// TIA Portal project "KWT_80413" (V14)

(* hardware
DEVICE "S7-1200-Station_1"  S7-1200 Station
   slot 0: "Baugruppenträger_0"  S7-1200 Rack  Rack  V1.0
   slot 1: "PLC_1"  CPU 1212C AC/DC/Rly  6ES7 212-1BE40-0XB0  V4.2
   slot 2: "AQ 2x14BIT_1"  SM 1232 AQ2  6ES7 232-4HB32-0XB0  V2.0
   slot 3: "DI 16x24VDC_1"  6ES7 221-1BH32-0XB0  V2.0
DEVICE "HMI_1"  KTP1200 Basic PN
   slot 0: "KTP1200 Basic PN"  KTP1200 Basic PN  6AV2 123-2MB03-0AX0  14.0.1.0
   slot 1: "HMI_RT_1"  KTP1200 Basic PN  6AV2 123-2MB03-0AX0  14.0.1.0
   slot 5: "HMI_1.IE_CP_1"  PROFINET Interface  14.0.1.0
      slot 1: "PROFINET Schnittstelle_1"  PROFINET Interface
         slot 1: "Port_1"  Port
*)

// ===== PLC "PLC_1"  CPU 1212C AC/DC/Rly =====

VAR_GLOBAL   // PLC tag table "Standard-Variablentabelle"
   "System_Byte" AT %MB1 : Byte;
   "FirstScan" AT %M1.0 : Bool;
   "DiagStatusUpdate" AT %M1.1 : Bool;
   "AlwaysTRUE" AT %M1.2 : Bool;
   "AlwaysFALSE" AT %M1.3 : Bool;
   "Clock_Byte" AT %MB0 : Byte;
   "Clock_10Hz" AT %M0.0 : Bool;
   "Clock_5Hz" AT %M0.1 : Bool;
   "Clock_2.5Hz" AT %M0.2 : Bool;
   "Clock_2Hz" AT %M0.3 : Bool;
   "Clock_1.25Hz" AT %M0.4 : Bool;
   "Clock_1Hz" AT %M0.5 : Bool;
   "Clock_0.625Hz" AT %M0.6 : Bool;
   "Clock_0.5Hz" AT %M0.7 : Bool;
   "Pumpe 1" AT %Q0.0 : Bool;   // Pumpe 1, -102K1, -36K6, Werkskreislauf
   "Pumpe 2" AT %Q0.1 : Bool;   // Pumpe 2, -102K2, -38K6, Werkskreislauf
   "Pumpe 3" AT %Q0.2 : Bool;   // Pumpe 3, -102K3, -41K6, Kühlturmkreislauf
   "Pumpe 4" AT %Q0.3 : Bool;   // Pumpe 4, -102K4, -43K6, Kühlturmkreislauf
   "Ventilator 1" AT %Q0.4 : Bool;   // Ventilator 1, -102K5, -31G1
   "Ventilator 2" AT %Q0.5 : Bool;   // Ventilator 2, -102K6, -33G1
   "Vorlauftemperatur" AT %IW64 : Int;
   "Rücklauftemperatur" AT %IW66 : Int;
   "Störung Pumpe 1" AT %I0.0 : Bool;   // -36K3
   "Betrieb Pumpe 1" AT %I0.1 : Bool;   // -36K6
   "Störung Pumpe 2" AT %I0.2 : Bool;   // -38K3
   "Betrieb Pumpe 2" AT %I0.3 : Bool;   // -38K6
   "Störung Pumpe 3" AT %I0.4 : Bool;   // -41K3
   "Betrieb Pumpe 3" AT %I0.5 : Bool;   // -41K6
   "Störung Pumpe 4" AT %I0.6 : Bool;   // -43K3
   "Betrieb Pumpe 4" AT %I0.7 : Bool;   // -43K6
   "stetige Ansteuerung FU 1" AT %QW96 : Int;
   "stetige Ansteuerung FU 2" AT %QW98 : Int;
   "Störung  Ventilator 1" AT %I12.0 : Bool;
   "Betrieb Ventilator 1" AT %I12.1 : Bool;
   "Rep.-Schalter Ventilator 1" AT %I12.2 : Bool;   // -31K9
   "Störung Ventiator 2" AT %I12.3 : Bool;
   "Betrieb Ventilator 2" AT %I12.4 : Bool;
   "Rep.-Schalter Ventilator 2" AT %I12.5 : Bool;   // -33K9
   "Betrieb Heizpatrone 1" AT %I12.6 : Bool;   // -51K6
   "Störung STB Heizpatrone 1" AT %I12.7 : Bool;   // -51K5
   "Betrieb Heizpatrone 2" AT %I13.0 : Bool;   // -52K6
   "Störung STB Heizpatrone 2" AT %I13.1 : Bool;   // -52K5
   "Absalzanlage" AT %I13.2 : Bool;   // -X6 11
   "DI Reserve(2)" AT %I13.3 : Bool;   // -X6 13
   "ZU-Klappen 1 Auf" AT %I13.4 : Bool;
   "ZU-Klappen 2 Auf" AT %I13.5 : Bool;
   "DI Reserve(3)" AT %I13.6 : Bool;   // -X6 15
   "DI Reserve(4)" AT %I13.7 : Bool;   // -X6 17
END_VAR

VAR_GLOBAL   // PLC tag table "Test"
   "tPumpe1" AT %M100.0 : Bool;
   "tPumpe2" AT %M100.1 : Bool;
   "tPumpe1Störung" AT %M100.2 : Bool;
   "tPumpe1Betrieb" AT %M100.3 : Bool;
   "tPumpe2Störung" AT %M100.4 : Bool;
   "tPumpe2Betrieb" AT %M100.5 : Bool;
   "tPumpe3Betrieb" AT %M100.6 : Bool;
   "tPumpe4Betrieb" AT %M100.7 : Bool;
END_VAR

DATA_BLOCK "Auto_DB"   // DB1
{ S7_Optimized_Access := 'TRUE' }
VERSION : 0.1
// stored: InstanceOfName Auto
"Auto"
BEGIN
END_DATA_BLOCK

DATA_BLOCK "Werkskreislauf_DB"   // DB2
{ S7_Optimized_Access := 'TRUE' }
VERSION : 0.1
// stored: InstanceOfName Werkskreislauf
"Werkskreislauf"
BEGIN
END_DATA_BLOCK

DATA_BLOCK "Global-DB"   // DB3
{ S7_Optimized_Access := 'TRUE' }
VERSION : 0.1
   VAR
      Vorlauftemperatur : Real;
      Rücklauftemperatur : Real;
      Auto : Bool := true;
   END_VAR
BEGIN
END_DATA_BLOCK

DATA_BLOCK "Kühlturmkreislauf_DB"   // DB4
{ S7_Optimized_Access := 'TRUE' }
VERSION : 0.1
// stored: InstanceOfName Kühlturmkreislauf
"Kühlturmkreislauf"
BEGIN
END_DATA_BLOCK

DATA_BLOCK "Temperatur_DB"   // DB11
{ S7_Optimized_Access := 'TRUE' }
VERSION : 0.1
// stored: InstanceOfName Temperatur
"Temperatur"
BEGIN
END_DATA_BLOCK

DATA_BLOCK "Hand_DB"   // DB12
{ S7_Optimized_Access := 'TRUE' }
VERSION : 0.1
// stored: InstanceOfName Hand
"Hand"
BEGIN
END_DATA_BLOCK

// folder: System blocks/Program resources

DATA_BLOCK "IEC_Timer_0_DB"   // DB5
{ S7_Optimized_Access := 'TRUE' }
AUTHOR : Simatic
FAMILY : IEC
NAME : IEC_TMR
VERSION : 1.0
// stored: InstanceOfName IEC_TIMER
"IEC_TIMER"
BEGIN
END_DATA_BLOCK

DATA_BLOCK "IEC_Timer_0_DB_1"   // DB6
{ S7_Optimized_Access := 'TRUE' }
AUTHOR : Simatic
FAMILY : IEC
NAME : IEC_TMR
VERSION : 1.0
// stored: InstanceOfName IEC_TIMER
"IEC_TIMER"
BEGIN
END_DATA_BLOCK

DATA_BLOCK "IEC_Timer_0_DB_2"   // DB7
{ S7_Optimized_Access := 'TRUE' }
AUTHOR : Simatic
FAMILY : IEC
NAME : IEC_TMR
VERSION : 1.0
// stored: InstanceOfName IEC_TIMER
"IEC_TIMER"
BEGIN
END_DATA_BLOCK

DATA_BLOCK "IEC_Timer_0_DB_3"   // DB8
{ S7_Optimized_Access := 'TRUE' }
AUTHOR : Simatic
FAMILY : IEC
NAME : IEC_TMR
VERSION : 1.0
// stored: InstanceOfName IEC_TIMER
"IEC_TIMER"
BEGIN
END_DATA_BLOCK

DATA_BLOCK "IEC_Timer_0_DB_4"   // DB9
{ S7_Optimized_Access := 'TRUE' }
AUTHOR : Simatic
FAMILY : IEC
NAME : IEC_TMR
VERSION : 1.0
// stored: InstanceOfName IEC_TIMER
"IEC_TIMER"
BEGIN
END_DATA_BLOCK

DATA_BLOCK "IEC_Timer_0_DB_5"   // DB10
{ S7_Optimized_Access := 'TRUE' }
AUTHOR : Simatic
FAMILY : IEC
NAME : IEC_TMR
VERSION : 1.0
// stored: InstanceOfName IEC_TIMER
"IEC_TIMER"
BEGIN
END_DATA_BLOCK

// folder: (top level)

FUNCTION_BLOCK "Auto"   // FB1, FBD
{ S7_Optimized_Access := 'TRUE' }
VERSION : 0.1
   VAR
      static_Min : Real;
   END_VAR
   VAR RETAIN
      static_Max : Real := 27.0;
   END_VAR
   VAR_TEMP
      temp_ret_val : Int;
      temp_dtl_out : DTL;
      temp_strang : Bool;
   END_VAR
BEGIN

REGION Network 1 (SCL)
   #temp_ret_val := RD_SYS_T(#temp_dtl_out);
   #temp_strang := #temp_dtl_out.DAY MOD 2 = 0;
END_REGION

REGION Network 2
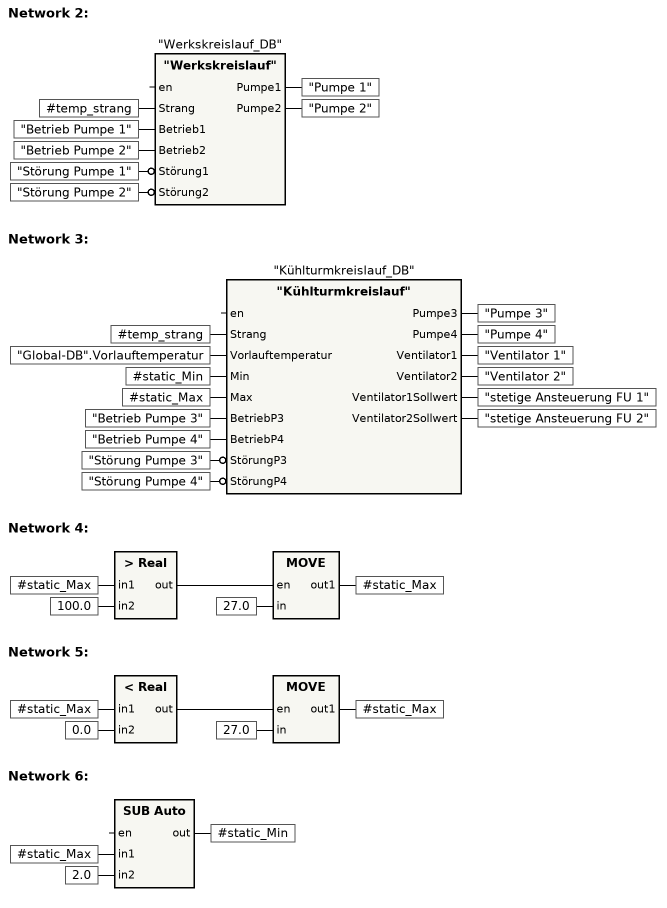
   "Werkskreislauf_DB"(Strang := #temp_strang,   // "Werkskreislauf"
                       Betrieb1 := "Betrieb Pumpe 1",
                       Betrieb2 := "Betrieb Pumpe 2",
                       Störung1 := NOT "Störung Pumpe 1",
                       Störung2 := NOT "Störung Pumpe 2",
                       Pumpe1 => "Pumpe 1",
                       Pumpe2 => "Pumpe 2");
END_REGION

REGION Network 3
   "Kühlturmkreislauf_DB"(Strang := #temp_strang,   // "Kühlturmkreislauf"
                          Vorlauftemperatur := "Global-DB".Vorlauftemperatur,
                          Min := #static_Min,
                          Max := #static_Max,
                          BetriebP3 := "Betrieb Pumpe 3",
                          BetriebP4 := "Betrieb Pumpe 4",
                          StörungP3 := NOT "Störung Pumpe 3",
                          StörungP4 := NOT "Störung Pumpe 4",
                          Pumpe3 => "Pumpe 3",
                          Pumpe4 => "Pumpe 4",
                          Ventilator1 => "Ventilator 1",
                          Ventilator2 => "Ventilator 2",
                          Ventilator1Sollwert => "stetige Ansteuerung FU 1",
                          Ventilator2Sollwert => "stetige Ansteuerung FU 2");
END_REGION

REGION Network 4
   IF #static_Max > 100.0 THEN #static_Max := 27.0; END_IF;
END_REGION

REGION Network 5
   IF #static_Max < 0.0 THEN #static_Max := 27.0; END_IF;
END_REGION

REGION Network 6
   #static_Min := #static_Max - 2.0;
END_REGION
END_FUNCTION_BLOCK

FUNCTION_BLOCK "Werkskreislauf"   // FB2, FBD
{ S7_Optimized_Access := 'TRUE' }
VERSION : 0.1
   VAR_INPUT
      Strang : Bool;
      Betrieb1 : Bool;
      Betrieb2 : Bool;
      Störung1 : Bool;
      Störung2 : Bool;
   END_VAR
   VAR_OUTPUT
      Pumpe1 : Bool;
      Pumpe2 : Bool;
   END_VAR
   VAR
      static_Pumpe1 : Bool;
      static_Pumpe2 : Bool;
      static_Nachlaufzeit : Time := T#10s;
   END_VAR
BEGIN

REGION Network 1
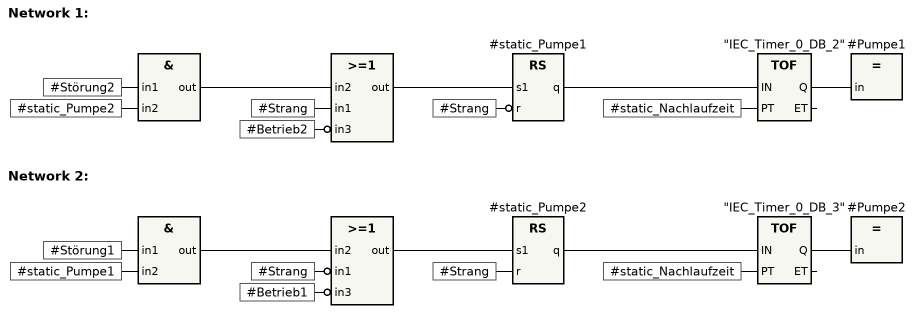
   IF NOT #Strang THEN
       #static_Pumpe1 := FALSE;   // RS flip-flop
   END_IF;
   IF (#Störung2 AND #static_Pumpe2) OR #Strang OR NOT #Betrieb2 THEN #static_Pumpe1 := TRUE; END_IF;
   "IEC_Timer_0_DB_2".TOF(IN := #static_Pumpe1, PT := #static_Nachlaufzeit);
   #Pumpe1 := "IEC_Timer_0_DB_2".Q;
END_REGION

REGION Network 2
   IF #Strang THEN
       #static_Pumpe2 := FALSE;   // RS flip-flop
   END_IF;
   IF (#Störung1 AND #static_Pumpe1) OR NOT #Strang OR NOT #Betrieb1 THEN #static_Pumpe2 := TRUE; END_IF;
   "IEC_Timer_0_DB_3".TOF(IN := #static_Pumpe2, PT := #static_Nachlaufzeit);
   #Pumpe2 := "IEC_Timer_0_DB_3".Q;
END_REGION
END_FUNCTION_BLOCK

FUNCTION_BLOCK "Kühlturmkreislauf"   // FB3, FBD
{ S7_Optimized_Access := 'TRUE' }
VERSION : 0.1
   VAR_INPUT
      Strang : Bool;
      Vorlauftemperatur : Real;
      Min : Real;
      Max : Real;
      BetriebP3 : Bool;
      BetriebP4 : Bool;
      StörungP3 : Bool;
      StörungP4 : Bool;
   END_VAR
   VAR_OUTPUT
      Pumpe3 : Bool;
      Pumpe4 : Bool;
      Ventilator1 : Bool;
      Ventilator2 : Bool;
      Ventilator1Sollwert : Int;
      Ventilator2Sollwert : Int;
   END_VAR
   VAR
      static_Pumpe3 : Bool;
      static_Pumpe4 : Bool;
      static_zu_kalt : Bool;
      static_zu_warm : Bool;
      static_Sollwert : Int;
      static_Ventilator_pt : Time := T#30s;
      static_Beide_Pumpen : Bool;
      static_Nachlaufzeit : Time := T#10s;
      "static_Max+1" : Real;
   END_VAR
   VAR_TEMP
      temp_norm_out : Real;
   END_VAR
BEGIN

REGION Network 1
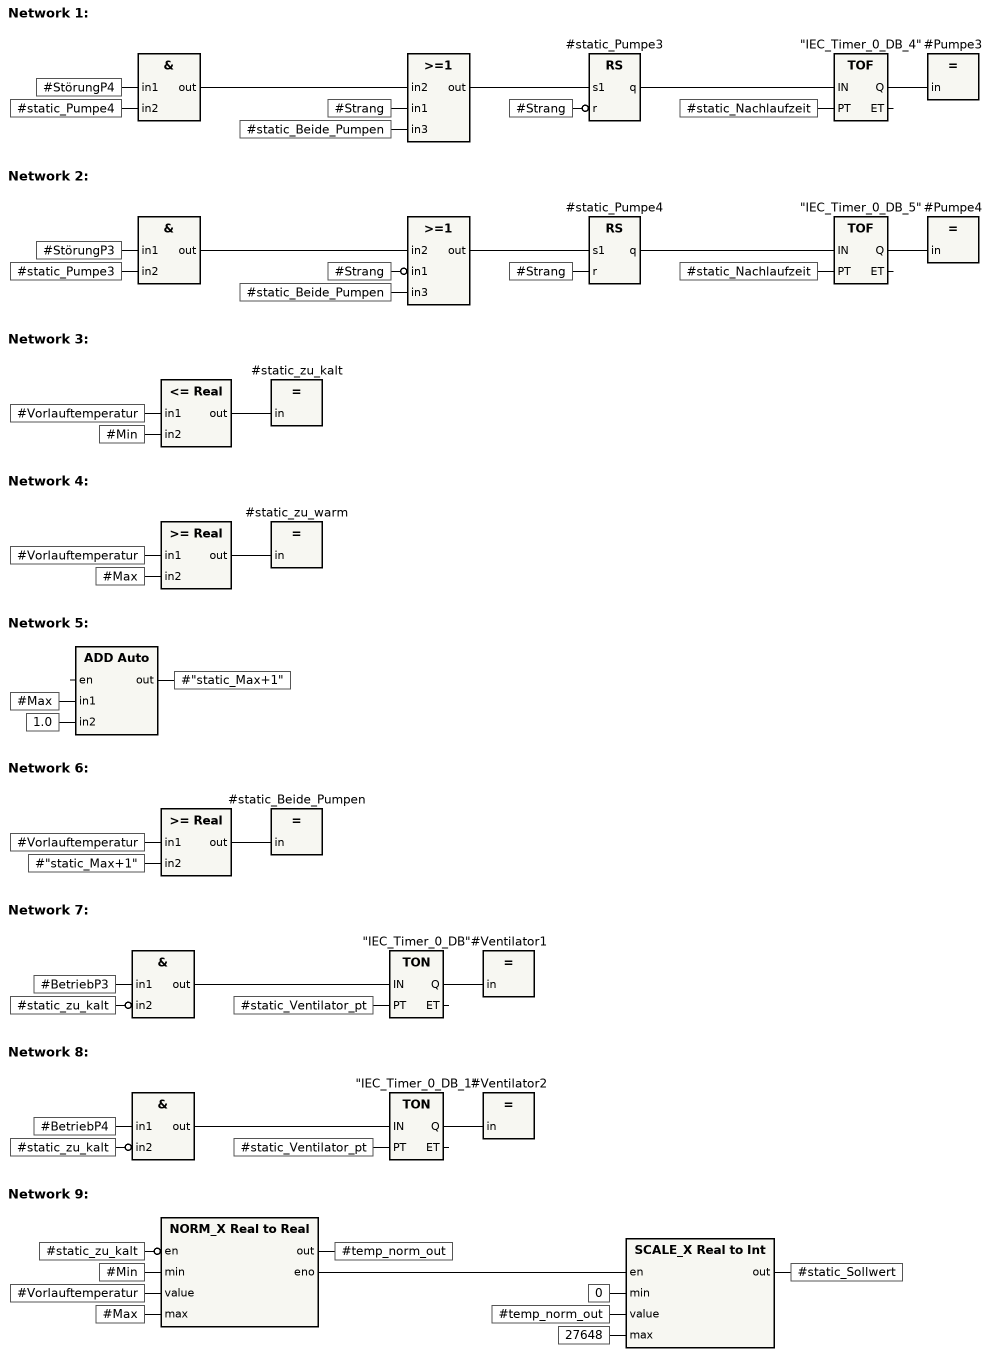
   IF NOT #Strang THEN
       #static_Pumpe3 := FALSE;   // RS flip-flop
   END_IF;
   IF (#StörungP4 AND #static_Pumpe4) OR #Strang OR #static_Beide_Pumpen THEN #static_Pumpe3 := TRUE; END_IF;
   "IEC_Timer_0_DB_4".TOF(IN := #static_Pumpe3, PT := #static_Nachlaufzeit);
   #Pumpe3 := "IEC_Timer_0_DB_4".Q;
END_REGION

REGION Network 2
   IF #Strang THEN
       #static_Pumpe4 := FALSE;   // RS flip-flop
   END_IF;
   IF (#StörungP3 AND #static_Pumpe3) OR NOT #Strang OR #static_Beide_Pumpen THEN
       #static_Pumpe4 := TRUE;
   END_IF;
   "IEC_Timer_0_DB_5".TOF(IN := #static_Pumpe4, PT := #static_Nachlaufzeit);
   #Pumpe4 := "IEC_Timer_0_DB_5".Q;
END_REGION

REGION Network 3
   #static_zu_kalt := #Vorlauftemperatur <= #Min;
END_REGION

REGION Network 4
   #static_zu_warm := #Vorlauftemperatur >= #Max;
END_REGION

REGION Network 5
   #"static_Max+1" := #Max + 1.0;
END_REGION

REGION Network 6
   #static_Beide_Pumpen := #Vorlauftemperatur >= #"static_Max+1";
END_REGION

REGION Network 7
   "IEC_Timer_0_DB".TON(IN := #BetriebP3 AND NOT #static_zu_kalt, PT := #static_Ventilator_pt);
   #Ventilator1 := "IEC_Timer_0_DB".Q;
END_REGION

REGION Network 8
   "IEC_Timer_0_DB_1".TON(IN := #BetriebP4 AND NOT #static_zu_kalt, PT := #static_Ventilator_pt);
   #Ventilator2 := "IEC_Timer_0_DB_1".Q;
END_REGION

REGION Network 9
   IF NOT #static_zu_kalt THEN
       #temp_norm_out := NORM_X(MIN := #Min, VALUE := #Vorlauftemperatur, MAX := #Max);
       #static_Sollwert := SCALE_X(MIN := 0, VALUE := #temp_norm_out, MAX := 27648);
   END_IF;
END_REGION

REGION Network 10
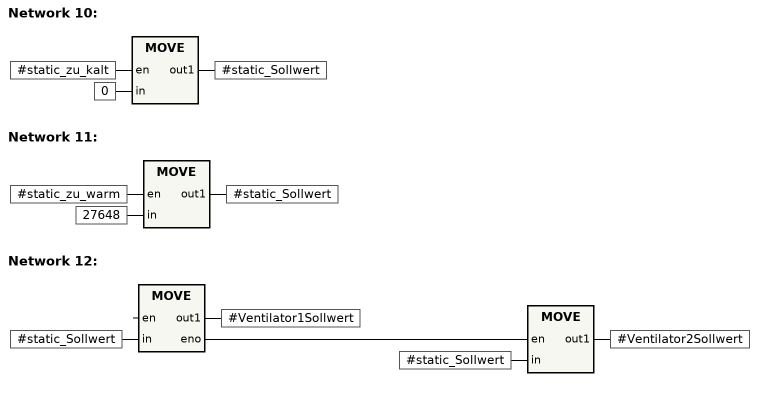
   IF #static_zu_kalt THEN #static_Sollwert := 0; END_IF;
END_REGION

REGION Network 11
   IF #static_zu_warm THEN #static_Sollwert := 27648; END_IF;
END_REGION

REGION Network 12
   #Ventilator1Sollwert := #static_Sollwert;
   #Ventilator2Sollwert := #static_Sollwert;
END_REGION
END_FUNCTION_BLOCK

FUNCTION_BLOCK "Temperatur"   // FB4, FBD
{ S7_Optimized_Access := 'TRUE' }
VERSION : 0.1
   VAR_INPUT
      IN_Vorlauftemp : Int;
      IN_Rücklauftemp : Int;
   END_VAR
   VAR_OUTPUT
      OUT_Vorlauftemp : Real;
      OUT_Rücklauftemp : Real;
   END_VAR
   VAR
      static_Vorlauftemp : Real;
      static_Rücklauftemp : Real;
   END_VAR
   VAR_TEMP   // added for the SCL form of the ladder/FBD networks
      _w1 : Bool;
   END_VAR
BEGIN

REGION Network 1
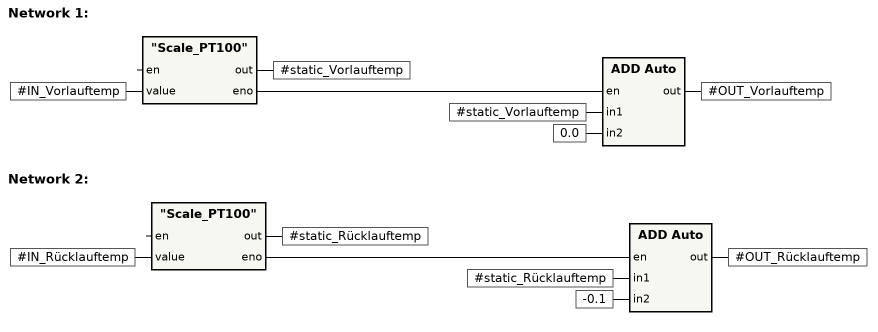
   "Scale_PT100"(value := #IN_Vorlauftemp, out => #static_Vorlauftemp, ENO => #_w1);
   IF #_w1 THEN #OUT_Vorlauftemp := #static_Vorlauftemp + 0.0; END_IF;
END_REGION

REGION Network 2
   "Scale_PT100"(value := #IN_Rücklauftemp, out => #static_Rücklauftemp, ENO => #_w1);
   IF #_w1 THEN #OUT_Rücklauftemp := #static_Rücklauftemp + (-0.1); END_IF;
END_REGION
END_FUNCTION_BLOCK

FUNCTION_BLOCK "Hand"   // FB5, FBD
{ S7_Optimized_Access := 'TRUE' }
VERSION : 0.1
   VAR
      "static_Vent1Soll%" : Int;
      "static_Vent2Soll%" : Int;
      static_Vent1Soll : Real;
      static_Vent2Soll : Real;
   END_VAR
   VAR_TEMP
      akk : Int;
   END_VAR
BEGIN

REGION Network 1
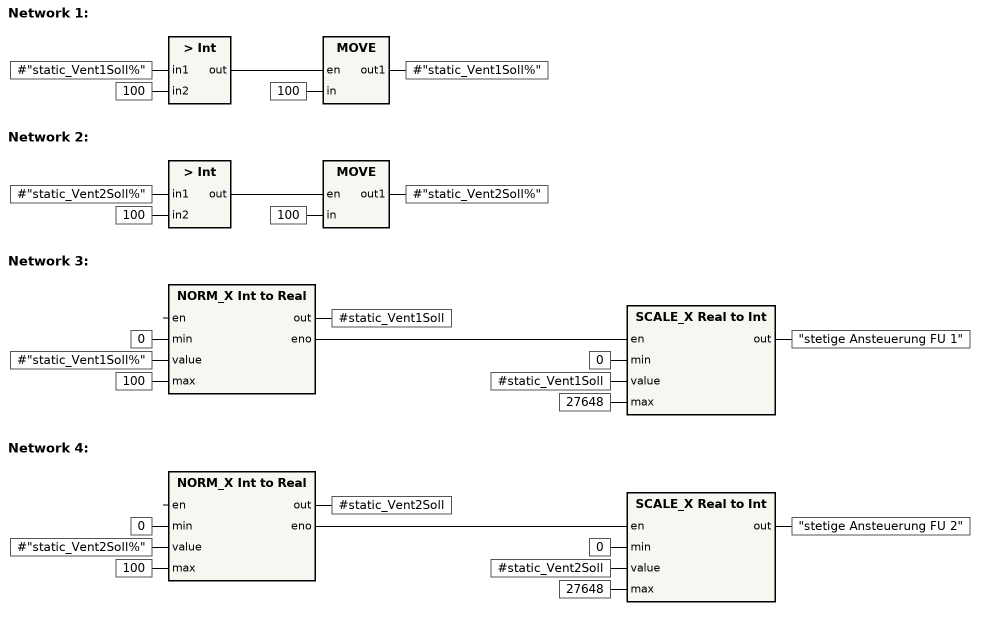
   IF #"static_Vent1Soll%" > 100 THEN #"static_Vent1Soll%" := 100; END_IF;
END_REGION

REGION Network 2
   IF #"static_Vent2Soll%" > 100 THEN #"static_Vent2Soll%" := 100; END_IF;
END_REGION

REGION Network 3
   #static_Vent1Soll := NORM_X(MIN := 0, VALUE := #"static_Vent1Soll%", MAX := 100);
   "stetige Ansteuerung FU 1" := SCALE_X(MIN := 0, VALUE := #static_Vent1Soll, MAX := 27648);
END_REGION

REGION Network 4
   #static_Vent2Soll := NORM_X(MIN := 0, VALUE := #"static_Vent2Soll%", MAX := 100);
   "stetige Ansteuerung FU 2" := SCALE_X(MIN := 0, VALUE := #static_Vent2Soll, MAX := 27648);
END_REGION
END_FUNCTION_BLOCK

FUNCTION "Scale_PT100" : Void   // FC1, FBD
{ S7_Optimized_Access := 'TRUE' }
VERSION : 0.1
   VAR_INPUT
      value : Int;
   END_VAR
   VAR_OUTPUT
      out : Real;
   END_VAR
   VAR_TEMP
      temp_norm_out : Real;
   END_VAR
BEGIN

REGION Network 1
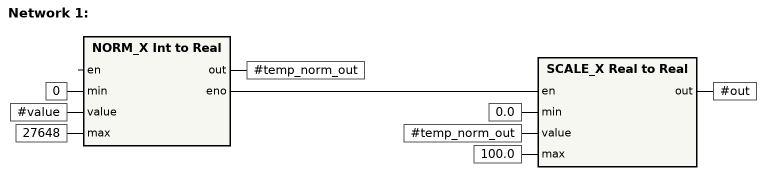
   #temp_norm_out := NORM_X(MIN := 0, VALUE := #value, MAX := 27648);
   #out := SCALE_X(MIN := 0.0, VALUE := #temp_norm_out, MAX := 100.0);
END_REGION
END_FUNCTION

ORGANIZATION_BLOCK "Main"   // OB1, FBD, ProgramCycle
TITLE = "Main Program Sweep (Cycle)"
{ S7_Optimized_Access := 'TRUE' }
VERSION : 0.1
   VAR_INPUT
      Initial_Call : Bool;   // Initial call of this OB
      Remanence : Bool;   // =True, if remanent data are available
   END_VAR
BEGIN

REGION Network 1
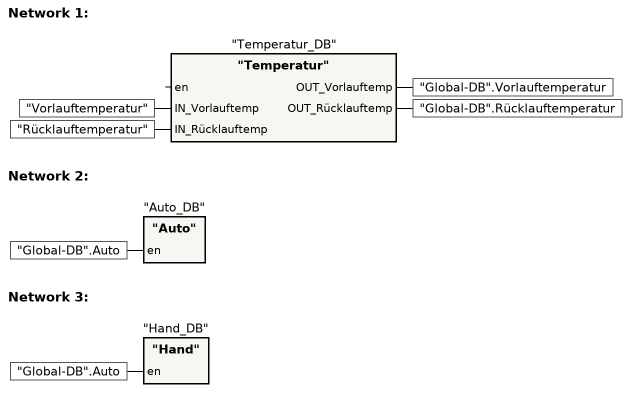
   "Temperatur_DB"(IN_Vorlauftemp := "Vorlauftemperatur",   // "Temperatur"
                   IN_Rücklauftemp := "Rücklauftemperatur",
                   OUT_Vorlauftemp => "Global-DB".Vorlauftemperatur,
                   OUT_Rücklauftemp => "Global-DB".Rücklauftemperatur);
END_REGION

REGION Network 2
   IF "Global-DB".Auto THEN
       "Auto_DB"();   // "Auto"
   END_IF;
END_REGION

REGION Network 3
   IF "Global-DB".Auto THEN
       "Hand_DB"();   // "Hand"
   END_IF;
END_REGION
END_ORGANIZATION_BLOCK

(* ===== HMI "HMI_RT_1" =====
system functions are stored by id; their names below are inferred from use
connection "HMI_Verbindung_1": ETHERNET, SMART_S7_1200_OMS

HMI tags "Standard-Variablentabelle"
   "Variable_Bildnummer" : UInt, internal
   "Global-DB_Vorlauftemperatur" : Real = PLC "Global-DB".Vorlauftemperatur, 1 s
   "Global-DB_Rücklauftemperatur" : Real = PLC "Global-DB".Rücklauftemperatur, 1 s
   "Global-DB_Auto" : Bool = PLC "Global-DB".Auto, 1 s
   "Pumpe 1" : Bool = PLC "Pumpe 1" AT %Q0.0, 1 s
   "Pumpe 2" : Bool = PLC "Pumpe 2" AT %Q0.1, 1 s
   "Pumpe 3" : Bool = PLC "Pumpe 3" AT %Q0.2, 1 s
   "Pumpe 4" : Bool = PLC "Pumpe 4" AT %Q0.3, 1 s
   "Ventilator 1" : Bool = PLC "Ventilator 1" AT %Q0.4, 1 s
   "Ventilator 2" : Bool = PLC "Ventilator 2" AT %Q0.5, 1 s
   "Hand_DB_static_Vent1Soll%" : Int = PLC Hand_DB.static_Vent1Soll%, 1 s
   "Hand_DB_static_Vent2Soll%" : Int = PLC Hand_DB.static_Vent2Soll%, 1 s
   "Auto_DB_static_Max" : Real = PLC Auto_DB.static_Max, 1 s

text list "Textliste_Bildnamen": 1 'Grundbild'

Template "Vorlage_1" 1280x800
   Button "Beenden" at 1182,752 size 67x47; TextOff 'Beenden'; PictureOff "ExitRuntime_KTP1200_Basic_PN_TR"; PictureOn "ExitRuntime_KTP1200_Basic_PN_TR"
      on Release: StopRuntime(0)
   Button "Template_Button" at 1054,752 size 67x47; TextOff 'Text'
   Button "Template_Button_1" at 926,752 size 67x47; TextOff 'Text'
   Button "Template_Button_2" at 798,752 size 67x47; TextOff 'Text'
   Button "Template_Button_3" at 670,752 size 67x47; TextOff 'Text'
   Button "Template_Button_4" at 542,752 size 67x47; TextOff 'Text'
   Button "Template_Button_5" at 414,752 size 67x47; TextOff 'Text'
   Button "Template_Button_6" at 286,752 size 67x47; TextOff 'Text'
   Button "Meldungen" at 158,752 size 67x47; TextOff 'Meldungen'; PictureOff "AlarmDisplay_KTP1200_Basic_PN_TR"; PictureOn "AlarmDisplay_KTP1200_Basic_PN_TR"
      on Release: function_ef3f5d25("Meldefenster_Nichtquittiert", -1)
   Button "Startbild" at 30,752 size 67x47; TextOff 'Startbild'; PictureOff "NavigateHome_KTP1200_Basic_PN_TR"; PictureOn "NavigateHome_KTP1200_Basic_PN_TR"
      on Release: ActivateScreen("Grundbild", 0)
   SymbolicIOField "Symbolisches_EA_Feld_Bild" at 87,9 size 1086x30; TextOff '0'; TextOn '1'; TextList "Textliste_Bildnamen"
      ProcessValue <- "Variable_Bildnummer"
      on Change: ActivateScreenByNumber("Variable_Bildnummer", 0)
   DateTimeField "HmiScreenItemData" at 1175,24 size 105x24
   DateTimeField "HmiScreenItemData_1" at 1175,0 size 105x24
   GraphicView "Logo" at 0,0 size 85x48; Picture "Logo von HMI_1"

screen "Grundbild" 1280x800, template "Vorlage_1"
   on GenerateScreen: SetTag("Variable_Bildnummer", 1)
   TextField "Textfeld_1" at 150,133 size 154x25; Text 'flow temperature'
   IOField "EA-Feld_1" at 326,133 size 96x32; FormatPattern s999999999.99
      ProcessValue <- "Global-DB_Vorlauftemperatur"
   TextField "Textfeld_2" at 3,46 size 150x94; Text 'Debrecen hűtőtorony +mező1'
   TextField "Textfeld_3" at 150,171 size 169x25; Text 'return temperature'
   IOField "EA-Feld_2" at 326,171 size 96x32; FormatPattern s999999999.99
      ProcessValue <- "Global-DB_Rücklauftemperatur"
   TextField "Textfeld_4" at 424,133 size 25x25; Text '°C'
   TextField "Textfeld_5" at 424,171 size 25x25; Text '°C'
   TrendView "Kurvenanzeige_1" at 153,428 size 600x300
   Switch "Schalter_1" at 633,133 size 120x32; CaptionText 'Switch'; TextOff 'HAND'; TextOn 'AUTO'
      ProcessValue <- "Global-DB_Auto"
   TextField "Textfeld_6" at 821,139 size 80x25; Text 'Pumpe 1'
      Visibility <- "Global-DB_Auto"
   Switch "Schalter_2" at 938,136 size 64x32; CaptionText 'Switch'; TextOff 'OFF'; TextOn 'ON'
      Visibility <- "Global-DB_Auto"
      ProcessValue <- "Pumpe 1"
   TextField "Textfeld_7" at 821,178 size 80x25; Text 'Pumpe 2'
      Visibility <- "Global-DB_Auto"
   Switch "Schalter_3" at 938,176 size 64x32; TextOn 'ON'; CaptionText 'Switch'; TextOff 'OFF'
      Visibility <- "Global-DB_Auto"
      ProcessValue <- "Pumpe 2"
   Switch "Schalter_4" at 938,216 size 64x32; TextOn 'ON'; CaptionText 'Switch'; TextOff 'OFF'
      Visibility <- "Global-DB_Auto"
      ProcessValue <- "Pumpe 3"
   Switch "Schalter_5" at 938,256 size 64x32; TextOn 'ON'; CaptionText 'Switch'; TextOff 'OFF'
      Visibility <- "Global-DB_Auto"
      ProcessValue <- "Pumpe 4"
   Switch "Schalter_6" at 938,296 size 64x32; TextOn 'ON'; CaptionText 'Switch'; TextOff 'OFF'
      Visibility <- "Global-DB_Auto"
      ProcessValue <- "Ventilator 1"
   Switch "Schalter_7" at 938,336 size 64x32; TextOn 'ON'; CaptionText 'Switch'; TextOff 'OFF'
      Visibility <- "Global-DB_Auto"
      ProcessValue <- "Ventilator 2"
   TextField "Textfeld_8" at 821,218 size 80x25; Text 'Pumpe 3'
      Visibility <- "Global-DB_Auto"
   TextField "Textfeld_9" at 821,260 size 80x25; Text 'Pumpe 4'
      Visibility <- "Global-DB_Auto"
   TextField "Textfeld_10" at 821,299 size 105x25; Text 'Ventilator 1'
      Visibility <- "Global-DB_Auto"
   TextField "Textfeld_11" at 821,340 size 105x25; Text 'Ventilator 1'
      Visibility <- "Global-DB_Auto"
   IOField "EA-Feld_3" at 1008,296 size 50x32; FormatPattern 999
      ProcessValue <- "Hand_DB_static_Vent1Soll%"
      Visibility <- "Global-DB_Auto"
   IOField "EA-Feld_4" at 1008,336 size 50x32; FormatPattern 999
      Visibility <- "Global-DB_Auto"
      ProcessValue <- "Hand_DB_static_Vent2Soll%"
   IOField "EA-Feld_5" at 326,211 size 96x32; FormatPattern s999999999.99
      ProcessValue <- "Auto_DB_static_Max"
   TextField "Textfeld_12" at 424,213 size 213x25; Text '°C default value is 27 °C'
   TextField "Textfeld_13" at 153,211 size 76x25; Text 'setpoint'
*)